KUKA KRL program: C3BI_JOG.src

&ACCESS RV
DEF C3BI_JOG( )
BAS (#INITMOV, 0)
PTP $AXIS_ACT

$BASE = {X 0.0, Y 0.0, Z 0.0, A 0.0, B 0.0, C 0.0}
$TOOL = {X 0.0, Y 0.0, Z 0.0, A 0.0, B 0.0, C 0.0}

C3BI_JOG_FRAME = {X 0.0, Y 0.0, Z 0.0, A 0.0, B 0.0, C 0.0}

$ADVANCE = 3

LOOP
CONTINUE
PTP_REL C3BI_JOG_FRAME C_PTP
ENDLOOP

END
